# EPICS StreamDevice protocol: ned/protocol/snshv.proto
Terminator = CR;
ReplyTimeout = 1000;
LockTimeout = 5000;
ReadTimeout  = 100;

read_voltage {
    out "?LV";
    in "?LV%05d";
}

write_voltage {
    out "*#%05d";
    in "*#%05d";
}
